FUNCTION_BLOCK FINAL FB_Safety
VAR_INPUT
	bEmergencyStopOK				AT%I*	: BOOL;
END_VAR
VAR_OUTPUT
END_VAR
VAR
END_VAR

END_FUNCTION_BLOCK

(* stored: Version 1.1.0.1, ProductVersion 3.1.4024.12
   POU FB_Safety: Id {ffbfa9ce-8ba4-405c-8606-945cde52289d}, SpecialFunc None *)
